// TIA Portal V19 export
FUNCTION_BLOCK "TYPIC_C106_IF_NET"   // FB82, FBD
TITLE = TYPIC_C106_IF_NET: Netaansluiting
{ S7_Optimized_Access := 'TRUE' }
AUTHOR : OCOTECH
FAMILY : Typical
NAME : C106.705
// Logisch Object Besturing: C106.705
// 
// De interne functie netaansluiting verzorgt de bewaking van een netaansluiting.
// stored: MemoryReserve 10, SetENOAutomatically false
   VAR_INPUT
      EXT_AUT { ExternalAccessible := 'False'; ExternalVisible := 'False'; ExternalWritable := 'False'} : Bool;   // Externe (hoofd) beveiliging (1 = OK)
      EXT_HW { ExternalAccessible := 'False'; ExternalVisible := 'False'; ExternalWritable := 'False'} : Bool;   // Sturings hardware (PLC) bewaking (1 = OK)
      IN_STO_NOK { ExternalAccessible := 'False'; ExternalVisible := 'False'; ExternalWritable := 'False'} : Bool;   // Storing aanwezig die niet observeerbaar tot gevolg heeft
      IN_STO_OK { ExternalAccessible := 'False'; ExternalVisible := 'False'; ExternalWritable := 'False'} : Bool;   // Storing aanwezig die observeerbaarheid niet beinvloed
      IN_NET_BSC1 { ExternalAccessible := 'False'; ExternalVisible := 'False'; ExternalWritable := 'False'} : Bool;   // Netaansluiting beschikbaar
      IN_NET_BSC2 { ExternalAccessible := 'False'; ExternalVisible := 'False'; ExternalWritable := 'False'} : Bool;   // Netaansluiting niet beschikbaar
      IN_NET_BSC3 { ExternalAccessible := 'False'; ExternalVisible := 'False'; ExternalWritable := 'False'} : Bool;   // Netaansluiting beperkt beschikbaar
      IN_STS_KR { ExternalAccessible := 'False'; ExternalVisible := 'False'; ExternalWritable := 'False'} : Bool;   // Kritiek
      IN_STS_GKR { ExternalAccessible := 'False'; ExternalVisible := 'False'; ExternalWritable := 'False'} : Bool;   // Gestopt kritiek
      IN_TYD_GKR { ExternalAccessible := 'False'; ExternalVisible := 'False'; ExternalWritable := 'False'} : Real;   // Tijdverloop voor Gestopt Kritiek
      IN_AUT_C106 { ExternalAccessible := 'False'; ExternalVisible := 'False'; ExternalWritable := 'False'} : Bool;   // Beveiligingen: serie geschakelde terugmelding (1 = OK)
   END_VAR
   VAR_OUTPUT
      VAR_IF_NET { ExternalAccessible := 'False'; ExternalVisible := 'False'; ExternalWritable := 'False'} : "C106_VAR_IF_NET_TYPIC";   // Struct met alle variabelen naar bovenliggende functies
   END_VAR
   VAR
      STO { ExternalWritable := 'False'} : Struct   // Storingen
         A001 : Bool;   // Beveiliging aangesproken
         A002 : Bool;   // Netaansluiting in storing
         A003 : Bool;   // Algemene storing netaansluiting
         A004 : Bool;   // Geen netaansluiting beschikbaar
         A005 : Bool;   // NSA niet gestart na uitval netaansluiting
      END_STRUCT;
      VAR { ExternalWritable := 'False'} : Struct   // Variabelen
         BSC1 { ExternalAccessible := 'False'; ExternalVisible := 'False'} : Bool;   // Netaansluiting beschikbaar
         BSC2 { ExternalAccessible := 'False'; ExternalVisible := 'False'} : Bool;   // Netaansluiting niet beschikbaar
         BSC3 { ExternalAccessible := 'False'; ExternalVisible := 'False'} : Bool;   // Netaansluiting beperkt beschikbaar
         STS_KR { ExternalAccessible := 'False'; ExternalVisible := 'False'} : Bool;   // Kritiek
         STS_GKR { ExternalAccessible := 'False'; ExternalVisible := 'False'} : Bool;   // Gestopt kritiek
         TYD_GKR { ExternalAccessible := 'False'; ExternalVisible := 'False'} : Real;   // Tijdverloop voor Gestopt Kritiek
         EXT_AUT { ExternalAccessible := 'False'; ExternalVisible := 'False'} : Bool;   // Externe (hoofd) beveiliging aangesproken
         EXT_HW { ExternalAccessible := 'False'; ExternalVisible := 'False'} : Bool;   // Sturings hardware (PLC) in storing
      END_STRUCT;
   END_VAR
BEGIN

REGION Network 1: START
END_REGION

REGION Network 2: +++ Verwerking meetwaarden en statussen +++
   // De meetwaarde en status wordt ontvangen vanuit de interne sturing.
END_REGION

REGION Network 3: +++ Storingen +++
   // Verwerken van de storingsmeldingen (inputs).
END_REGION

REGION Network 4: Storing A001: Beveiliging aangesproken
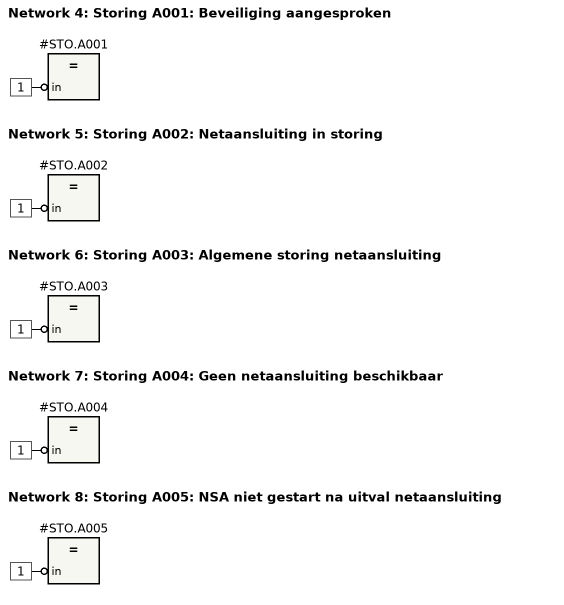
   #STO.A001 := NOT 1;
END_REGION

REGION Network 5: Storing A002: Netaansluiting in storing
   #STO.A002 := NOT 1;
END_REGION

REGION Network 6: Storing A003: Algemene storing netaansluiting
   #STO.A003 := NOT 1;
END_REGION

REGION Network 7: Storing A004: Geen netaansluiting beschikbaar
   #STO.A004 := NOT 1;
END_REGION

REGION Network 8: Storing A005: NSA niet gestart na uitval netaansluiting
   #STO.A005 := NOT 1;
END_REGION

REGION Network 9 (SCL): EINDE
   // Variabelen van intern scada rakvlak naar outputs copieren
   #VAR_IF_NET.BSC1 := #VAR.BSC1;
   #VAR_IF_NET.BSC2 := #VAR.BSC2;
   #VAR_IF_NET.BSC3 := #VAR.BSC3;
   #VAR_IF_NET.STS_KR := #VAR.STS_KR;
   #VAR_IF_NET.STS_GKR := #VAR.STS_GKR;
   #VAR_IF_NET.TYD_GKR := #VAR.TYD_GKR;
   #VAR_IF_NET.EXT_AUT := #VAR.EXT_AUT;
   #VAR_IF_NET.EXT_HW := #VAR.EXT_HW;
   #VAR_IF_NET.STO := #STO;
END_REGION
END_FUNCTION_BLOCK
